FUNCTION_BLOCK DisableConveyor
  (* Standard: 61499-2 *)
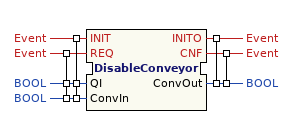
  EVENT_INPUT
    INIT WITH QI, ConvIn;
    REQ WITH QI, ConvIn;
  END_EVENT
  EVENT_OUTPUT
    INITO WITH ConvOut;
    CNF WITH ConvOut;
  END_EVENT
  VAR_INPUT
    QI : BOOL;
    ConvIn : BOOL;
  END_VAR
  VAR_OUTPUT
    ConvOut : BOOL;
  END_VAR
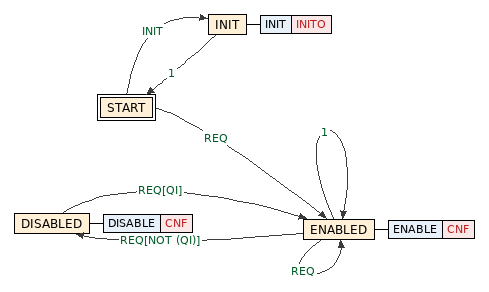
  EC_STATES
    START;
    INIT : INIT -> INITO;
    ENABLED : ENABLE -> CNF;
    DISABLED : DISABLE -> CNF;
  END_STATES
  EC_TRANSITIONS
    START TO INIT := INIT;
    INIT TO START := 1;
    ENABLED TO DISABLED := REQ[NOT (QI)];
    START TO ENABLED := REQ;
    DISABLED TO ENABLED := REQ[QI];
    ENABLED TO ENABLED := REQ;
    ENABLED TO ENABLED := 1;
  END_TRANSITIONS
  ALGORITHM INIT IN ST:

  END_ALGORITHM
  ALGORITHM ENABLE IN ST:
ConvOut := ConvIn;&#10;
  END_ALGORITHM
  ALGORITHM DISABLE IN ST:
ConvOut := FALSE;&#10;
  END_ALGORITHM
END_FUNCTION_BLOCK
